FUNCTION_BLOCK FB_VisuControl EXTENDS FB_UniversalVisu
VAR
END_VAR

bBackupRestoreDisabled := TRUE;
SUPER^();

METHOD PROTECTED  MS_Emergency
;
END_METHOD

END_FUNCTION_BLOCK

(* stored: Version 1.1.0.1, ProductVersion 3.1.4024.9
   POU FB_VisuControl: Id {0bfae5f4-05f6-4ba2-8d1c-2f6d5de3971a}, SpecialFunc None
   Method MS_Emergency: Id {2a34c643-f64a-4582-8b3a-6c75d3cb4aac} *)
